        // Enable remaining temperature controls
        nott_t_ctrls.tc_sidecar.M_SetEnable();
        nott_t_ctrls.tc_photonic_chip.M_SetEnable();
        nott_t_ctrls.tc_base_plate.M_SetEnable();
        nott_t_ctrls.tc_shields.M_SetEnable();

        // Set warm-up setpoints
        nott_t_ctrls.tc_detector.M_Set_SetPoint(
            m_eSetpointType    := E_METIS_CTRL_SETPOINT_SWITCH.FIXED,
            m_lrFixedSetpoint  := cfg.lrTemp_Det,
            m_lrSetpointOffset := 0.0,
            m_pSetpointTemp    := nott_temps.M_SetTemperatureSensor(0)
        );

        nott_t_ctrls.tc_detector_spare.M_Set_SetPoint(
            m_eSetpointType    := E_METIS_CTRL_SETPOINT_SWITCH.FIXED,
            m_lrFixedSetpoint  := cfg.lrTemp_Det,
            m_lrSetpointOffset := 0.0,
            m_pSetpointTemp    := nott_temps.M_SetTemperatureSensor(0)
        );

        nott_t_ctrls.tc_sidecar.M_Set_SetPoint(
            m_eSetpointType    := E_METIS_CTRL_SETPOINT_SWITCH.FIXED,
            m_lrFixedSetpoint  := cfg.lrTemp_Sidecar,
            m_lrSetpointOffset := 0.0,
            m_pSetpointTemp    := nott_temps.M_SetTemperatureSensor(0)
        );

        nott_t_ctrls.tc_photonic_chip.M_Set_SetPoint(
            m_eSetpointType    := E_METIS_CTRL_SETPOINT_SWITCH.FIXED,
            m_lrFixedSetpoint  := cfg.lrTemp_PhotonicChip, 
            m_lrSetpointOffset := 0.0,
            m_pSetpointTemp    := nott_temps.M_SetTemperatureSensor(0)
        );

        nott_t_ctrls.tc_base_plate.M_Set_SetPoint(
            m_eSetpointType    := E_METIS_CTRL_SETPOINT_SWITCH.FIXED,
            m_lrFixedSetpoint  := cfg.lrTemp_BasePlate,
            m_lrSetpointOffset := 0.0,
            m_pSetpointTemp    := nott_temps.M_SetTemperatureSensor(0)
        );

        nott_t_ctrls.tc_shields.M_Set_SetPoint(
            m_eSetpointType    := E_METIS_CTRL_SETPOINT_SWITCH.FIXED,
            m_lrFixedSetpoint  := cfg.lrTemp_Shield,
            m_lrSetpointOffset := 0.0,
            m_pSetpointTemp    := nott_temps.M_SetTemperatureSensor(0)
        );

        stat.sState  := 'WARMING UP';
        stat.sStatus := 'Warm-up heaters enabled';

        stat.nState := E_NOTT_CRYO_WARMUP_STATE.WARMING_UP;


    E_NOTT_CRYO_WARMUP_STATE.WARMING_UP:

        out_bPermit_Evacuation_Stop := FALSE;
        out_bPermit_CoolDown        := FALSE;

        IF NOT in_bEnable THEN
            stat.nState := E_NOTT_CRYO_WARMUP_STATE.STOP_WARMUP;

        ELSIF nott_temps.out_bHighestTempValid
              AND (nott_temps.out_lrHighestTemp > cfg.lrTemp_HighLimit) THEN

            stat.bError := TRUE;
            stat.sErrorText := CONCAT('High temperature limit exceeded at ', nott_temps.out_sHighestTempName);
            stat.sStatus := stat.sErrorText;
            stat.nState := E_NOTT_CRYO_WARMUP_STATE.STOP_WARMUP;

        ELSIF bAllWarm THEN
            stat.nState := E_NOTT_CRYO_WARMUP_STATE.WARM_TEMPERATURE_ACHIEVED;
            stat.sStatus := 'Warm temperature achieved';

        ELSE
            stat.sStatus := 'Warming up...';
        END_IF;


    E_NOTT_CRYO_WARMUP_STATE.WARM_TEMPERATURE_ACHIEVED:

        IF in_bEnable THEN
            stat.sState  := 'WARM';
            stat.sStatus := 'Warm temperature achieved';

            out_bPermit_Evacuation_Stop := TRUE;
            out_bPermit_CoolDown        := TRUE;

            // Keep temperature control active at warm targets
        ELSE
            stat.nState := E_NOTT_CRYO_WARMUP_STATE.STOP_WARMUP;
        END_IF;


    E_NOTT_CRYO_WARMUP_STATE.STOP_WARMUP:

        out_bPermit_Evacuation_Stop := FALSE;
        out_bPermit_CoolDown        := FALSE;

        nott_heaters.h_detector.M_SetDisable();
        nott_heaters.h_detector_spare.M_SetDisable();
        nott_heaters.h_sidecar.M_SetDisable();
        nott_heaters.h_photonic_chip.M_SetDisable();
        nott_heaters.h_base_plate.M_SetDisable();
        nott_heaters.h_shield.M_SetDisable();

        nott_t_ctrls.tc_detector.M_SetDisable();
        nott_t_ctrls.tc_detector_spare.M_SetDisable();
        nott_t_ctrls.tc_sidecar.M_SetDisable();
        nott_t_ctrls.tc_photonic_chip.M_SetDisable();
        nott_t_ctrls.tc_base_plate.M_SetDisable();
        nott_t_ctrls.tc_shields.M_SetDisable();

        stat.bActive := FALSE;
        stat.sState  := 'OFF';
        stat.sStatus := 'Warm-up stopped';

        stat.nState := E_NOTT_CRYO_WARMUP_STATE.OFF;


ELSE
    stat.bError := TRUE;
    stat.sErrorText := 'Unknown warm-up state';
    stat.sStatus := stat.sErrorText;
    stat.nState := E_NOTT_CRYO_WARMUP_STATE.NONE;
END_CASE;

M_StateMachine := TRUE;
END_METHOD

METHOD M_UpdateStatus : BOOL
VAR_INPUT
END_VAR
stat.bEnabled		:= in_bEnable;
END_METHOD

END_FUNCTION_BLOCK

// ---- POUs/Routines/Evacuation/FB_NOTT_CRYO_EVAC.TcPOU
FUNCTION_BLOCK FB_NOTT_CRYO_EVAC EXTENDS FB_CRYO_EVAC_BASE_50
VAR_INPUT
END_VAR
VAR
	//
	// Pumps
	//
	{attribute 'TcHmiSymbol.Show'}
	pump_pvp:	FB_NOTT_PUMP_HICUBE_80_NEO;	// Pre-vacuum Pump
	{attribute 'TcHmiSymbol.Show'}
	pump_tmp:	FB_NOTT_PUMP_HIPACE80;	// Turbo Molecular Pump
	
	{attribute 'TcHmiSymbol.Show'}
	bPermitStart:	BOOL := FALSE;
	{attribute 'TcHmiSymbol.Show'}
	bPermitStop:	BOOL := FALSE;
	{attribute 'TcHmiSymbol.Show'}
	{attribute 'TcHmiSymbol.ReadOnly'}	
	bEvacuationActive:		BOOL := FALSE;			// Flag if controller is ACTIVE
	{attribute 'TcHmiSymbol.Show'}
	{attribute 'TcHmiSymbol.ReadOnly'}	
	bEmergency:		BOOL := FALSE;			// Vacuum Emergency
	
	// Power for pressure sensors (TODO)
	q_bPower_VAG1	AT %Q*:	BOOL := TRUE;
	q_bPower_VAGC	AT %Q*:	BOOL := TRUE;
	
	// Control via DIs for Pumps (DI access request)
	q_bDIsCtrl_PVP	AT %Q*:	BOOL := TRUE;
	q_bDIsCtrl_TMP	AT %Q*:	BOOL := TRUE;
	
	// Rotation speed setting mode for pumps (DI1)
	q_bRotSpeedMode_PVP	AT %Q*:	BOOL := TRUE;
	q_bRotSpeedMode_TMP	AT %Q*:	BOOL := TRUE;
	
	// Pressure valve PVV1 power
	q_bPower_PVV1	AT %Q*:	BOOL := TRUE;
	// Pressure valve PVV1 OFF Flag
	q_bPVV1_OFF_Flag	AT %Q*:	BOOL := TRUE;

	// Testing
	sDevId:	STRING := '001';
	bUpdateCmds_PVP:	BOOL;
	bUpdateCmds_TMP:	BOOL;

// NOTT-specific evacuation pressure-rise safety
tonPressureRiseWindow: TON;
bPressureRiseWindowInit: BOOL := FALSE;
bPressureRiseEvacRestarted: BOOL := FALSE;
lrPressureRiseStart: LREAL := 0.0;
lrPressureRiseDelta: LREAL := 0.0;
bPressureRiseSafetyArmed: BOOL := FALSE;
	
END_VAR

SUPER^();

// M_Configure();

// Testing: to be removed
//
// Change pump RS-485 Device ID on the fly.
M_UpdatePumpCommands();

// M_ExecuteControllers();

q_bPVV1_OFF_Flag := NOT PVV1.Actuator.q_bCtrl;

CASE stat.nState	OF
		E_CRYO_EVAC_STATE_50.NONE:
			bEvacuationActive	:= FALSE;
		
		E_CRYO_EVAC_STATE_50.OFF:
			bEvacuationActive	:= FALSE;
	ELSE
		
		bEvacuationActive		:= TRUE;
END_CASE

METHOD M_Configure
VAR_INPUT
END_VAR
VAR
	tpCfgRef:	REFERENCE TO T_NOTT_PUMP_HIPACE80_CFG;
END_VAR
//
// Specific PDS IR Imager configuration.
//
IF NOT stat.bConfigured	THEN
	//
	// MANDATORY !!!
	// Call base FB::M_Configure() to set the pointers.
	//
	SUPER^.M_Configure();
	

	// MANDATORY: Set References for pumps!!!
	// If not done, system will crash !!!
	pvpRef	REF=pump_pvp;
	tmpRef	REF=pump_tmp;
	

	// Specific instance configuration, e.g. anything different
	// from the default values given in the cfg structure 
	// of type T_CRYO_EVAC_CFG_50.
	//
	// Set pressure sensor type
	cfg.nType_VAG1	:= E_CRYO_SENSOR_TYPE_PRESS.PKR_360;
	
	// Set pressure threshold for starting TMP after opening PVV1.
	
	cfg.lrThld_TMP_after_PVV1	:= 4.8;	
	
	// Set timeout for stopping turbo pump to 15 min (900000 ms)
	tpCfgRef	REF=pump_tmp.cfg;
	tpCfgRef.nTimeoutStart	:= 900000;
	tpCfgRef.nTimeoutStop	:= 900000;


	stat.bConfigured	:= TRUE;
END_IF
END_METHOD

METHOD M_ExecuteControllers
VAR_INPUT
END_VAR
//
// Specific PDS IR Imager HW.
//

// Roughing Pump
ctrl.cor_PVP(in_bEnable:=ctrl.bEnable_PVP);	// Command override

pump_pvp(	
	in_bSimulation	:= FALSE,
	in_sName		:= 'PVP',
	in_bEnable		:= ctrl.cor_PVP.out_bEnable,
	in_nModel		:= 30,
	in_bAutoMonitor	:= TRUE,
	in_sCmdSuffix:= '$R',
	in_sReplySuffix:= '$R',
	in_nPeriod		:= 3000);

// Turbo Molecular Pump
ctrl.cor_TMP(in_bEnable:=ctrl.bEnable_TMP);	// Command override

pump_tmp(	
	in_bSimulation	:= FALSE,
	in_sName		:= 'TMP',
	in_bEnable		:= ctrl.cor_TMP.out_bEnable,
	in_nModel		:= 30,
	in_bAutoMonitor	:= TRUE,
	in_nPeriod		:= 3000,
	in_sCmdSuffix:= '$R',
	in_sReplySuffix:= '$R');


// Valves are controlled in the base FB
SUPER^.M_ExecuteControllers();
END_METHOD

METHOD M_PermitStart_Evacuation
VAR_INPUT
	in_bPermissionStart: BOOL;
END_VAR
bPermitStart := in_bPermissionStart;
END_METHOD

METHOD M_PermitStop_Evacuation
VAR_INPUT
	in_bPermissionStop: BOOL;
END_VAR
bPermitStop := in_bPermissionStop;
END_METHOD

METHOD M_SafetyCheck
VAR_INPUT
END_VAR
VAR CONSTANT
    lrPress_EmergencyReset : LREAL := 10.0E-1; // [mbar]
    lrPressRiseTrip        : LREAL := 5.0;     // [mbar rise in 10 seconds]
    tPressureRiseWindow    : TIME  := T#10S;
END_VAR
SUPER^.M_SafetyCheck();

IF NOT in_RefVAGC.stat.bValid THEN
    tonPressureRiseWindow(IN := FALSE);
    bPressureRiseWindowInit := FALSE;
    RETURN;
END_IF

// Arm this safety only after evacuation has once reached vacuum.
// This avoids false trips from noisy atmospheric-pressure readings.
IF NOT bPressureRiseSafetyArmed THEN
    tonPressureRiseWindow(IN := FALSE);
    bPressureRiseWindowInit := FALSE;

    IF bEvacuationActive
       AND (in_RefVAGC.stat.lrPressure < lrPress_EmergencyReset) THEN
        bPressureRiseSafetyArmed := TRUE;
    END_IF

    RETURN;
END_IF

// Emergency latch behavior.
IF stat.bEmergency THEN
    ctrl.bEnable_PVV1 := FALSE;
    stat.bWarning     := TRUE;

    IF in_RefVAGC.stat.lrPressure < lrPress_EmergencyReset THEN
        stat.bEmergency := FALSE;
        stat.bWarning   := FALSE;

        bPressureRiseEvacRestarted := FALSE;
        bPressureRiseWindowInit    := FALSE;
        tonPressureRiseWindow(IN := FALSE);

        // Keep armed, because we are still below the reset pressure.
        bPressureRiseSafetyArmed := TRUE;

        stat.sStatus := 'VAGC pressure below emergency reset threshold.';
    END_IF

    RETURN;
END_IF

// Normal armed monitoring.
IF NOT bPressureRiseWindowInit THEN
    lrPressureRiseStart := in_RefVAGC.stat.lrPressure;
    lrPressureRiseDelta := 0.0;
    bPressureRiseWindowInit := TRUE;
END_IF

tonPressureRiseWindow(IN := TRUE, PT := tPressureRiseWindow);

IF tonPressureRiseWindow.Q THEN
    lrPressureRiseDelta :=
        in_RefVAGC.stat.lrPressure - lrPressureRiseStart;

    IF (lrPressureRiseDelta >= lrPressRiseTrip)
       AND NOT bPressureRiseEvacRestarted THEN

        ctrl.bEnable_PVV1 := FALSE;

        stat.bEmergency := TRUE;
        stat.bWarning   := TRUE;

        bPressureRiseEvacRestarted := TRUE;

        // Replace with the correct base restart state.
        stat.nState := E_CRYO_EVAC_STATE_50.CLOSE_PVV1_START;

        stat.sStatus :=
            'Emergency: VAGC pressure rise > 5 mbar in 10 s. PVV1 closed, evacuation restarted.';
    END_IF

    IF NOT stat.bEmergency THEN
        tonPressureRiseWindow(IN := FALSE);
        bPressureRiseWindowInit := FALSE;
    END_IF
END_IF
END_METHOD

METHOD M_UpdatePumpCommands
VAR_INPUT
END_VAR
VAR
	i:			INT;
	refCfg:		REFERENCE TO T_CRYO_PUMP_SERIAL_CFG;
	refPump:	REFERENCE TO FB_CRYO_PUMP_SERIAL;
	strTmp:		STRING;	// New command string
	sCmd:		STRING;
END_VAR
IF bUpdateCmds_PVP  OR  bUpdateCmds_TMP THEN
	IF bUpdateCmds_PVP  THEN
		bUpdateCmds_PVP	:= FALSE;
		refCfg	REF=pump_pvp.cfg;
		refPump	REF=pump_pvp;
	ELSIF bUpdateCmds_TMP THEN
		bUpdateCmds_TMP	:= FALSE;
		refCfg	REF=pump_tmp.cfg;
		refPump	REF=pump_tmp;
	END_IF

	
	// Replace Device ID (first three chars) all INIT and READ commands.
	// NOTE: Commands already contain checksum in last 3 char.
	// We start from new Dev ID in the first 3 char and discard last 3 char.
	// Call to M_PVP_Checksum() will add the new checksum.
	// Skip empty commands
	FOR i:=1 TO 8 DO
		strTmp	:= sDevId;	// Start from the new ID that occupy 3 chars.
		sCmd	:= refCfg.cmdList_Init[i].cmd;
		IF sCmd <> '' THEN
			strTmp	:= CONCAT(strTmp, MID(sCmd, LEN(sCmd)-6, 4));
			refCfg.cmdList_Init[i].cmd	:= refPump.M_PVP_Checksum(strTmp);
		ELSE
			EXIT;
		END_IF
	END_FOR
	
	FOR i:=1 TO 16 DO
		strTmp	:= sDevId;	// Start from the new ID that occupy 3 chars.
		sCmd	:= refCfg.cmdList_Read[i].cmd;
		IF sCmd <> '' THEN
			strTmp	:= CONCAT(strTmp, MID(sCmd, LEN(sCmd)-6, 4));
			refCfg.cmdList_Read[i].cmd	:= refPump.M_PVP_Checksum(strTmp);
		ELSE
			EXIT;
		END_IF
	END_FOR
	
END_IF
END_METHOD

END_FUNCTION_BLOCK

// ---- POUs/Devices/ThermalBox/FB_NOTT_THERMAL_BOX_CONTROL.TcPOU
FUNCTION_BLOCK FB_NOTT_THERMAL_BOX_CONTROL
VAR_INPUT
	in_tCycleTime:	TIME := T#10MS;
END_VAR
VAR_IN_OUT
	{attribute 'OPC.UA.DA' := '0'}
	nott_temps:						FB_NOTT_TEMPERATURES;
	{attribute 'OPC.UA.DA' := '0'}
	nott_heaters:					FB_NOTT_HEATERS;
	{attribute 'OPC.UA.DA' := '0'}
	nott_t_ctrls:      				FB_NOTT_TCTRLs;
	{attribute 'OPC.UA.DA' := '0'}
	nott_t_votes: 					FB_NOTT_VOTERS;
END_VAR
VAR
// 	{attribute 'TcHmiSymbol.Show'}
// 	cfg:	T_NOTT_THERMAL_BOX_CFG;
// 	{attribute 'TcHmiSymbol.Show'}
// 	ctrl:	T_NOTT_THERMAL_BOX_CTRL;
// 	{attribute 'TcHmiSymbol.Show'}
// 	stat:	T_NOTT_THERMAL_BOX_STAT;

	{attribute 'TcHmiSymbol.Show'}
	tc_fan:		FB_NOTT_CTRL_TEMPERATURE;
	{attribute 'TcHmiSymbol.Show'}
	tc_valve:	FB_NOTT_CTRL_TEMPERATURE;
	{attribute 'TcHmiSymbol.Show'}
	fan:		FB_NOTT_FAN;
	{attribute 'TcHmiSymbol.Show'}
	valve:		FB_METIS_CONTROL_VALVE;

	bFanAutoReady:		BOOL;
	bValveAutoReady:	BOOL;
END_VAR

METHOD M_SetDisable
//ctrl.bEnable := FALSE;
END_METHOD

METHOD M_SetEnable
//ctrl.bEnable := TRUE;
END_METHOD

END_FUNCTION_BLOCK

// ---- POUs/Devices/Fans/FB_NOTT_FAN.TcPOU
FUNCTION_BLOCK FB_NOTT_FAN
VAR_INPUT
	in_sName:				STRING;
	in_sAutoSetpointSource:	STRING;
	in_lrAutoSetpointValue:	LREAL;		// Temperature-controller output [0..100 %]
	in_tCycleTime:			TIME := T#10MS;
END_VAR
VAR
	{attribute 'TcHmiSymbol.Show'}
	cfg:	T_NOTT_FAN_CFG;
	{attribute 'TcHmiSymbol.Show'}
	ctrl:	T_NOTT_FAN_CTRL;
	{attribute 'TcHmiSymbol.Show'}
	stat:	T_NOTT_FAN_STAT;

	// Link these process-image variables to the selected EL2535 and ES1084 channels.
	{attribute 'TcHmiSymbol.Show'}
	i_bTach AT %I*:	BOOL;
	{attribute 'TcHmiSymbol.Show'}
	q_nPwmCommand AT %Q*:	INT;

	rtrigTach:	R_TRIG;
	rtrigEnable:	R_TRIG;
	tonRpmWindow:	TON;
	tonNoTach:	TON;
	tonStartBoost:	TON;
	bStarting:	BOOL := FALSE;
	bTach:		BOOL := FALSE;
	lrDemand:	LREAL := 0.0;
	lrOutputDuty:	LREAL := 0.0;
	nWindowPulses:	UDINT := 0;
END_VAR

stat.sName := in_sName;
stat.sAutoSetpointSource := in_sAutoSetpointSource;

// The thermal-box controller must be configured reverse acting (negative Kp):
// fan demand increases when measured temperature rises above setpoint.
IF ctrl.bAuto THEN
	lrDemand := in_lrAutoSetpointValue;
ELSE
	lrDemand := ctrl.lrManualDutyPct;
END_IF

IF lrDemand < 0.0 THEN
	lrDemand := 0.0;
ELSIF lrDemand > 100.0 THEN
	lrDemand := 100.0;
END_IF
stat.lrDemandPct := lrDemand;

rtrigEnable(CLK := ctrl.bEnable AND (lrDemand > 0.0));
IF rtrigEnable.Q THEN
	bStarting := TRUE;
	tonStartBoost(IN := FALSE, PT := cfg.tStartBoost);
END_IF

IF NOT ctrl.bEnable OR (lrDemand <= 0.0) THEN
	bStarting := FALSE;
	tonStartBoost(IN := FALSE, PT := cfg.tStartBoost);
	stat.lrDutyPct := 0.0;
	stat.bActive := ctrl.bEnable;
ELSE
	stat.bActive := TRUE;

	IF bStarting THEN
		tonStartBoost(IN := TRUE, PT := cfg.tStartBoost);
		stat.lrDutyPct := cfg.lrStartDutyPct;
		IF tonStartBoost.Q THEN
			bStarting := FALSE;
			tonStartBoost(IN := FALSE, PT := cfg.tStartBoost);
		END_IF
	ELSE
		IF lrDemand <= 0.0 THEN
			stat.lrDutyPct := 0.0;
		ELSIF lrDemand < cfg.lrMinRunningDutyPct THEN
			stat.lrDutyPct := cfg.lrMinRunningDutyPct;
		ELSIF lrDemand > cfg.lrMaxDutyPct THEN
			stat.lrDutyPct := cfg.lrMaxDutyPct;
		ELSE
			stat.lrDutyPct := lrDemand;
		END_IF
	END_IF
END_IF

IF stat.lrDutyPct < 0.0 THEN
	stat.lrDutyPct := 0.0;
ELSIF stat.lrDutyPct > 100.0 THEN
	stat.lrDutyPct := 100.0;
END_IF

lrOutputDuty := stat.lrDutyPct;
IF cfg.bInvertPwmOutput THEN
	lrOutputDuty := 100.0 - lrOutputDuty;
END_IF
q_nPwmCommand := LREAL_TO_INT(lrOutputDuty * INT_TO_LREAL(cfg.nPwmFullScale) / 100.0);

// ES1084 tach input. The fan supplies two rising pulses per revolution.
bTach := i_bTach;
IF cfg.bInvertTachInput THEN
	bTach := NOT bTach;
END_IF
rtrigTach(CLK := bTach);

IF rtrigTach.Q THEN
	nWindowPulses := nWindowPulses + 1;
	stat.nPulseCount := stat.nPulseCount + 1;
END_IF

tonRpmWindow(IN := TRUE, PT := cfg.tRpmWindow);
IF tonRpmWindow.Q THEN
	IF cfg.nPulsesPerRevolution > 0 THEN
		stat.lrSpeedRpm :=
			UDINT_TO_LREAL(nWindowPulses) * 60.0
			/ UINT_TO_LREAL(cfg.nPulsesPerRevolution)
			/ (TIME_TO_LREAL(cfg.tRpmWindow) / 1000.0);
	ELSE
		stat.lrSpeedRpm := 0.0;
	END_IF
	nWindowPulses := 0;
	tonRpmWindow(IN := FALSE, PT := cfg.tRpmWindow);
END_IF

// Reset the no-tach timer on every observed pulse.
tonNoTach(
	IN := ctrl.bEnable
		AND (stat.lrDutyPct >= cfg.lrMinRunningDutyPct)
		AND NOT rtrigTach.Q,
	PT := cfg.tStallDelay);

stat.bStallAlarm := tonNoTach.Q;
stat.bRunning := ctrl.bEnable AND (stat.lrSpeedRpm > 0.0) AND NOT stat.bStallAlarm;

// At maximum fan speed the pulse period is about 7 ms. A 10 ms task can miss
// edges even before considering the ES1084 3 ms input filter.
stat.bTachMeasurementLimited := in_tCycleTime > T#2MS;

METHOD M_SetDisable
ctrl.bEnable := FALSE;
END_METHOD

METHOD M_SetEnable
ctrl.bEnable := TRUE;
END_METHOD

END_FUNCTION_BLOCK

// ---- GlobalTextList.TcGTLO
TEXTLIST GlobalTextList
  876 = '%.1f'
  866 = '%.2f'
  778 = '%d'
  154 = '%s'
  640 = 'Configuration'
  284 = 'Control Mode'
  439 = 'Ctrl Signal :'
  784 = 'Drive Elec. Hours :'
  133 = 'Drive Elec. Temp [°C] :'
  905 = 'Error :'
  325 = 'Error Status'
  386 = 'Failure/Error Core'
  837 = 'FW Version'
  1833 = 'FW Version :'
  981 = 'Gas Balast Valve'
  418 = 'Gas Ballast Valve Enable'
  116 = 'Gas Ballast valve status'
  110 = 'GroupBox'
  858 = 'HW Version'
  2127 = 'HW Version :'
  873 = 'ID'
  145 = 'If ON, control output signal is active.'
  81 = 'Initialized'
  257 = 'Motor Current [mA] :'
  157 = 'Motor Power [W] :'
  804 = 'Motor Voltage [V] :'
  396 = 'Nominal Speed [rpm] :'
  611 = 'OK for Process, i.e. speed ≥ nominal speed'
  413 = 'presence of a warning'
  172 = 'Pressure'
  186 = 'Pressure Gauge'
  407 = 'Pressure Raw '
  894 = 'Pressure Sensor '
  216 = 'Pressure Sensor Active'
  434 = 'Pressure Sensor ON'
  587 = 'Pressure Text'
  385 = 'Pump Hours :'
  1038 = 'pump speed > 0 rpm'
  1651 = 'Pump Speed [rpm] :'
  148 = 'Pump State'
  1668 = 'Pump Temp [°C] :'
  384 = 'Ready :'
  12 = 'Running :'
  16 = 'Sensor Failed'
  670 = 'Sensor State'
  19 = 'START'
  401 = 'Status'
  119 = 'STOP'
  935 = 'Venting Enable'
END_TEXTLIST

// ---- VISUs/GUI_TEMPLATE_HIPACE_80.TcVIS
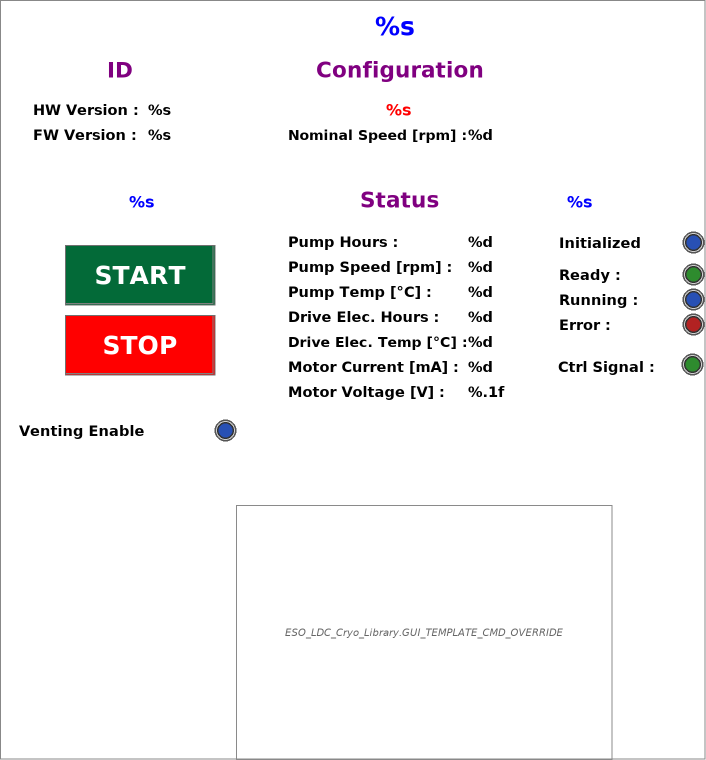
VISUALIZATION GUI_TEMPLATE_HIPACE_80  // 706x760
VAR_IN_OUT
	m_Instance:	FB_NOTT_PUMP_HIPACE80;
	m_bEnable:	BOOL;	// Flag to start/stop the pump
END_VAR
    Rectangle (45,55 150x30), "ID"
    Rectangle (310,55 180x30), "Configuration"
    Rectangle (325,185 150x30), "Status"
    Lamp1 (681,262 25x25), tooltip "OK for Process, i.e. speed ≥ nominal speed", variable: m_Instance.stat.bReady, style: Lamp-Lamp1-Green
    Lamp1 (681,287 25x25), tooltip "pump speed > 0 rpm", variable: m_Instance.stat.bMoving, style: Lamp-Lamp1-Blue
    Lamp1 (681,312 25x25), tooltip "presence of a warning", variable: m_Instance.stat.bFailure, style: Lamp-Lamp1-Red
    Rectangle (556,260 110x30), "Ready :"
    Rectangle (556,285 110x30), "Running :"
    Rectangle (556,310 110x30), "Error :"
    Rectangle (285,120 180x30), "Nominal Speed [rpm] :"
    Rectangle (285,227 180x30), "Pump Hours :"
    Rectangle (285,302 180x30), "Drive Elec. Hours :"
    Rectangle (465,120 70x30), "%d", text variable: m_Instance.stat.nNominalSpeed
    Rectangle (465,227 70x30), "%d", text variable: m_Instance.stat.nPumpHours
    Rectangle (465,302 70x30), "%d", text variable: m_Instance.stat.nElecHours
    Rectangle (285,252 180x30), "Pump Speed [rpm] :"
    Rectangle (465,252 70x30), "%d", text variable: m_Instance.stat.nPumpSpeed
    Rectangle (285,327 180x30), "Drive Elec. Temp [°C] :", text variable: m_Instance.stat.nElecTemp
    Rectangle (465,327 70x30), "%d", text variable: m_Instance.stat.nElecTemp
    Rectangle (285,277 180x30), "Pump Temp [°C] :"
    Rectangle (465,277 70x30), "%d", text variable: m_Instance.stat.nPumpTemp
    Rectangle (285,352 180x30), "Motor Current [mA] :", text variable: m_Instance.stat.nMotorCurr
    Rectangle (465,352 70x30), "%d", text variable: m_Instance.stat.nMotorCurr
    Rectangle (285,377 180x30), "Motor Voltage [V] :", text variable: m_Instance.stat.nMotorVolt
    Rectangle (465,377 70x30), "%.1f", text variable: m_Instance.stat.lrMotorVolt
    Rectangle (280,11 230x30), "%s", text variable: m_Instance.in_sName
    Rectangle (289,95 220x30), "%s", tooltip "Control Mode", text variable: m_Instance.stat.sCtrlMode
    Rectangle (145,95 130x30), "%s", tooltip "HW Version", text variable: m_Instance.stat.sHwVersion
    Rectangle (145,120 130x30), "%s", tooltip "FW Version", text variable: m_Instance.stat.sFwVersion
    Button (65,245 150x60), "START"
        OnMouseClick: execute { m_bEnable := TRUE; }
    Button (65,315 150x60), "STOP"
        OnMouseClick: execute { m_bEnable := FALSE; }
    Lamp1 (680,352 25x25), tooltip "If ON, control output signal is active.", variable: m_Instance.q_bStart, style: Lamp-Lamp1-Green
    Rectangle (555,352 110x30), "Ctrl Signal :"
    Rectangle (457,187 246x30), "%s", tooltip "Pump State", text variable: m_Instance.stat.sPumpState
    Rectangle (92,187 100x30), "%s", tooltip "Error Status", text variable: m_Instance.stat.sFailureCode
    Rectangle (30,95 110x30), "HW Version :"
    Rectangle (30,120 110x30), "FW Version :"
    Rectangle (556,228 110x30), "Initialized"
    Lamp1 (681,230 25x25), tooltip "OK for Process, i.e. speed ≥ nominal speed", variable: m_Instance.stat.bInitialised, style: Lamp-Lamp1-Blue
    Lamp1 (213,418 25x25), tooltip "OK for Process, i.e. speed ≥ nominal speed", variable: m_Instance.stat.bVentEnable, style: Lamp-Lamp1-Blue
    Rectangle (16,416 182x30), "Venting Enable"
    Frame (236,505 376x255)
        shows ESO_LDC_Cryo_Library.GUI_TEMPLATE_CMD_OVERRIDE(m_Cmd := MAIN.nott_cryo_ctrl.evac.ctrl.cor_TMP)
END_VISUALIZATION

// ---- VISUs/TEMPLATE_NOTT_PUMPS.TcVIS
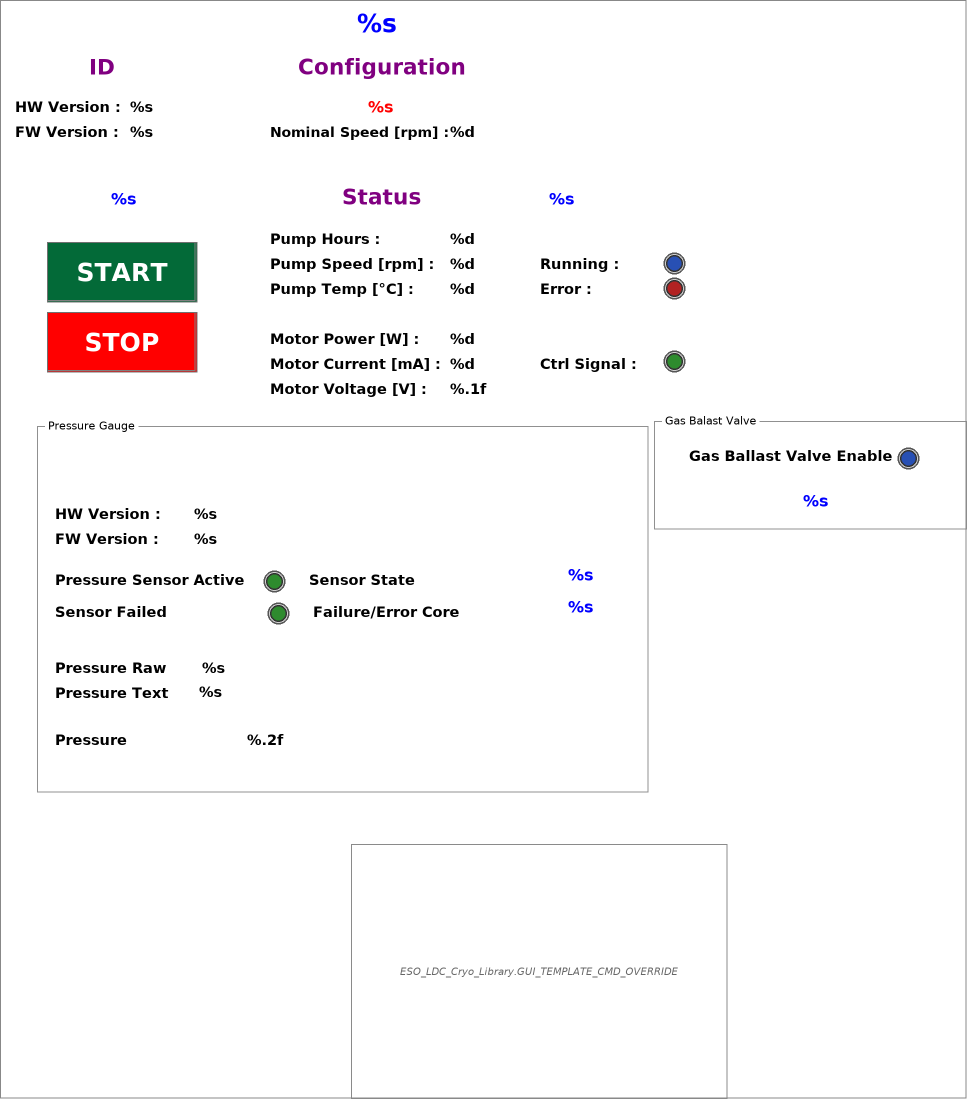
VISUALIZATION TEMPLATE_NOTT_PUMPS  // 967x1099
VAR_IN_OUT
	m_Instance:	FB_NOTT_PUMP_HICUBE_80_NEO;
	m_bEnable:	BOOL;	// Flag to start/stop the pump
	
END_VAR
    Rectangle (27,52 150x30), "ID"
    Rectangle (292,52 180x30), "Configuration"
    Rectangle (307,182 150x30), "Status"
    Lamp1 (662,251 25x25), tooltip "pump speed > 0 rpm", variable: m_Instance.stat.bMoving, style: Lamp-Lamp1-Blue
    Lamp1 (662,276 25x25), tooltip "presence of a warning", variable: m_Instance.stat.bFailure, style: Lamp-Lamp1-Red
    Rectangle (537,249 110x30), "Running :"
    Rectangle (537,274 110x30), "Error :"
    Rectangle (267,117 180x30), "Nominal Speed [rpm] :"
    Rectangle (267,224 180x30), "Pump Hours :"
    Rectangle (447,117 70x30), "%d", text variable: m_Instance.stat.nNominalSpeed
    Rectangle (447,224 70x30), "%d", text variable: m_Instance.stat.nPumpHours
    Rectangle (267,249 180x30), "Pump Speed [rpm] :"
    Rectangle (447,249 70x30), "%d", text variable: m_Instance.stat.nPumpSpeed
    Rectangle (267,274 180x30), "Pump Temp [°C] :"
    Rectangle (447,274 70x30), "%d", text variable: m_Instance.stat.nPumpTemp
    Rectangle (267,349 180x30), "Motor Current [mA] :"
    Rectangle (447,349 70x30), "%d", text variable: m_Instance.stat.nMotorCurr
    Rectangle (267,374 180x30), "Motor Voltage [V] :"
    Rectangle (447,374 70x30), "%.1f", text variable: m_Instance.stat.lrMotorVolt
    Rectangle (262,8 230x30), "%s", text variable: m_Instance.in_sName
    Rectangle (271,92 220x30), "%s", tooltip "Control Mode", text variable: m_Instance.stat.sCtrlViaInt
    Rectangle (127,92 130x30), "%s", tooltip "HW Version", text variable: m_Instance.stat.sHwVersion
    Rectangle (127,117 130x30), "%s", tooltip "FW Version", text variable: m_Instance.stat.sFwVersion
    Button (47,242 150x60), "START"
        OnMouseClick: execute { m_bEnable := TRUE; }
    Button (47,312 150x60), "STOP"
        OnMouseClick: execute { m_bEnable := FALSE; }
    Lamp1 (662,349 25x25), tooltip "If ON, control output signal is active.", variable: m_Instance.q_bStart, style: Lamp-Lamp1-Green
    Rectangle (537,349 110x30), "Ctrl Signal :"
    Rectangle (439,184 246x30), "%s", tooltip "Pump State", text variable: m_Instance.stat.sPumpState
    Rectangle (74,184 100x30), "%s", tooltip "Error Status", text variable: m_Instance.stat.sFailureCode
    Rectangle (267,324 180x30), "Motor Power [W] :"
    Rectangle (447,324 70x30), "%d", text variable: m_Instance.stat.nElecPower
    Rectangle (12,92 110x30), "HW Version :"
    Rectangle (12,117 110x30), "FW Version :"
    Frame (351,844 376x255)
        shows ESO_LDC_Cryo_Library.GUI_TEMPLATE_CMD_OVERRIDE(m_Cmd := MAIN.nott_cryo_ctrl.evac.ctrl.cor_PVP)
    GroupBox (37,418 611x374), "Pressure Gauge"
        Lamp1 (225,151 25x25), tooltip "Pressure Sensor ON", variable: m_Instance.stat.PresSens_bSensorOn, style: Lamp-Lamp1-Green
        Rectangle (15,147 254x30), "Pressure Sensor Active"
        Lamp1 (229,183 25x25), tooltip "Pressure Sensor ON", variable: m_Instance.stat.PresSens_bFailure, style: Lamp-Lamp1-Green
        Rectangle (269,147 254x30), "Sensor State"
        Rectangle (450,174 188x30), "%s", tooltip "Error Status", text variable: m_Instance.stat.PresSens_sFailureCode
        Rectangle (273,179 254x30), "Failure/Error Core"
        Rectangle (15,179 254x30), "Sensor Failed"
        Rectangle (450,142 188x30), "%s", tooltip "Error Status", text variable: m_Instance.stat.PresSens_sSensorState
        Rectangle (15,81 110x30), "HW Version :"
        Rectangle (154,81 130x30), "%s", tooltip "HW Version", text variable: m_Instance.stat.PresSens_sHwVersion
        Rectangle (154,106 130x30), "%s", tooltip "FW Version", text variable: m_Instance.stat.PresSens_sFwVersion
        Rectangle (15,106 110x30), "FW Version :"
        Rectangle (15,235 138x30), "Pressure Raw"
        Rectangle (162,235 130x30), "%s", tooltip "HW Version", text variable: m_Instance.stat.PresSens_sPressureRaw
        Rectangle (159,259 130x30), "%s", tooltip "FW Version", text variable: m_Instance.stat.PresSens_sPressureText
        Rectangle (15,260 142x30), "Pressure Text"
        Rectangle (15,307 180x30), "Pressure"
        Rectangle (207,307 197x30), "%.2f", text variable: m_Instance.stat.PresSens_lrPressure_hPa
    GroupBox (654,413 313x116), "Gas Balast Valve"
        Rectangle (39,73 246x30), "%s", tooltip "Gas Ballast valve status", text variable: m_Instance.stat.sGasBallastMode
        Lamp1 (242,33 25x25), tooltip "If ON, control output signal is active.", variable: m_Instance.stat.bGasBallastEnabled, style: Lamp-Lamp1-Blue
        Rectangle (32,28 211x30), "Gas Ballast Valve Enable"
END_VISUALIZATION

// ---- VISUs/VISU_BASE_PLATE_HTR.TcVIS
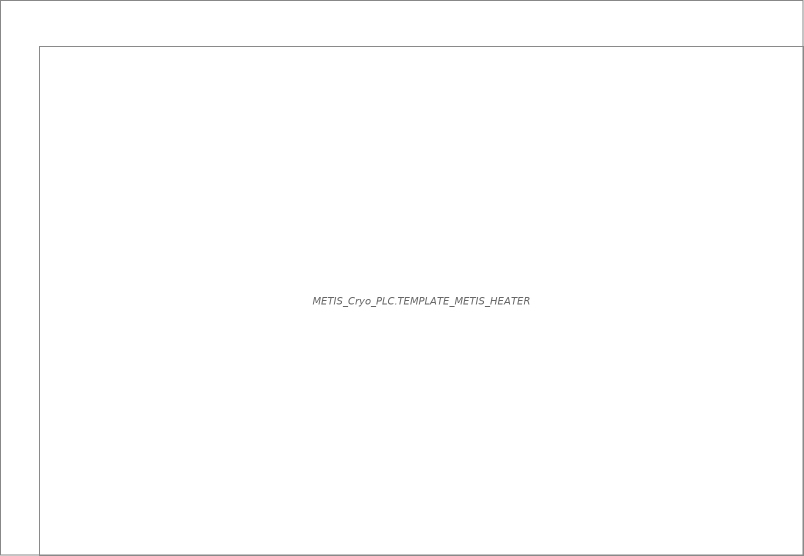
VISUALIZATION VISU_BASE_PLATE_HTR  // 804x556
    Frame (39,46 765x510)
        shows METIS_Cryo_PLC.TEMPLATE_METIS_HEATER(m_instance := MAIN.nott_cryo_ctrl.nott_heaters.h_base_plate)
END_VISUALIZATION

// ---- VISUs/VISU_Detector_Heater.TcVIS
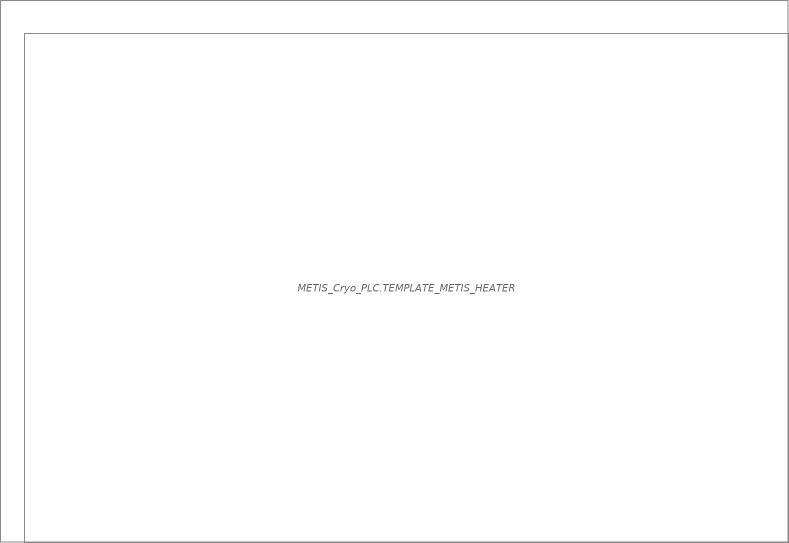
VISUALIZATION VISU_Detector_Heater  // 789x543
    Frame (24,33 765x510)
        shows METIS_Cryo_PLC.TEMPLATE_METIS_HEATER(m_instance := MAIN.nott_cryo_ctrl.nott_heaters.h_detector)
END_VISUALIZATION

// ---- VISUs/VISU_NOTT_PRESSURES.TcVIS
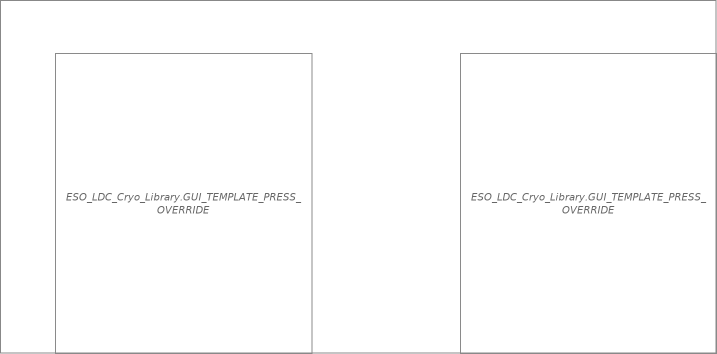
VISUALIZATION VISU_NOTT_PRESSURES  // 717x354
    Frame (55,53 257x301)
        shows ESO_LDC_Cryo_Library.GUI_TEMPLATE_PRESS_OVERRIDE(m_Cmd := MAIN.nott_cryo_ctrl.ctrl.por_VAGC, m_Press := MAIN.nott_cryo_ctrl.VAGC)
    Frame (460,53 257x301)
        shows ESO_LDC_Cryo_Library.GUI_TEMPLATE_PRESS_OVERRIDE(m_Cmd := MAIN.nott_cryo_ctrl.ctrl.por_HPG, m_Press := MAIN.nott_cryo_ctrl.HPG)
END_VISUALIZATION

// ---- VISUs/VISU_NOTT_RP.TcVIS
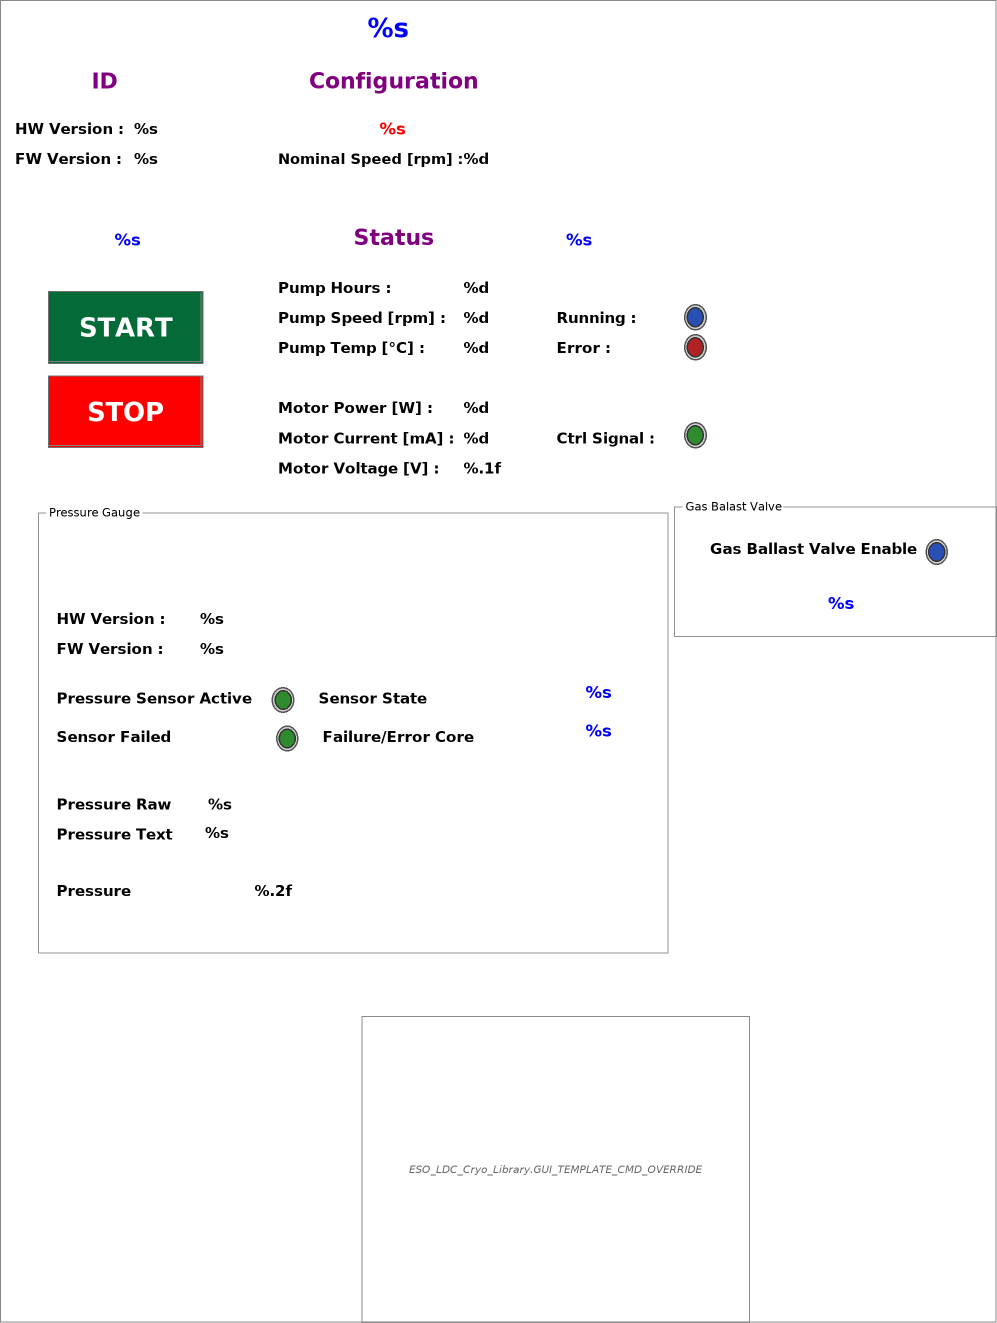
VISUALIZATION VISU_NOTT_RP  // 997x1323
    Frame (0,0 997x1323)
        shows TEMPLATE_NOTT_PUMPS(m_Instance := MAIN.nott_cryo_ctrl.evac.pump_pvp)
END_VISUALIZATION

// ---- VISUs/VISU_NOTT_TP.TcVIS
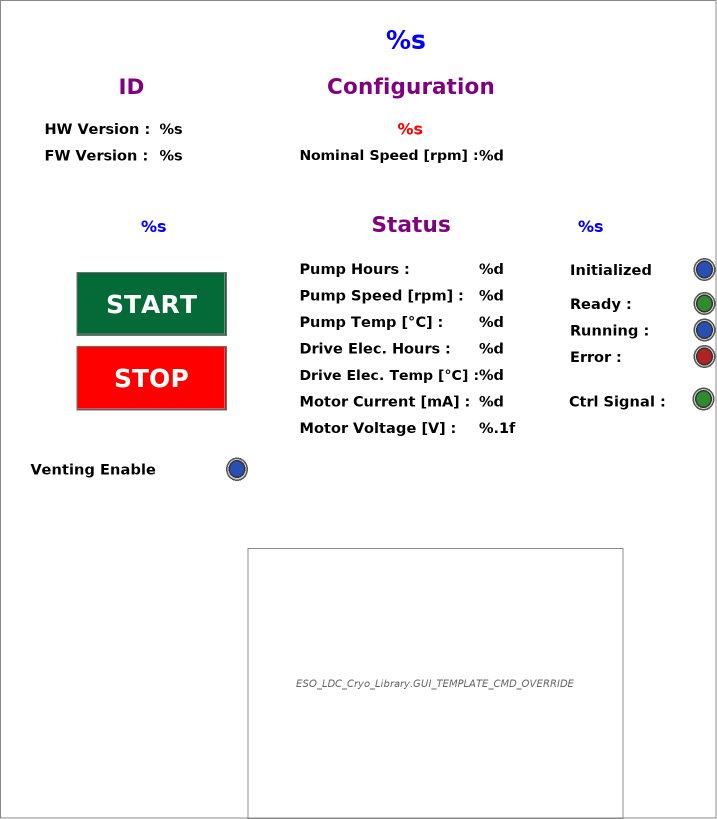
VISUALIZATION VISU_NOTT_TP  // 717x819
    Frame (12,12 705x807)
        shows GUI_TEMPLATE_HIPACE_80(m_Instance := MAIN.nott_cryo_ctrl.evac.pump_tmp)
END_VISUALIZATION

// ---- VISUs/VISU_PTC_COOLER.TcVIS
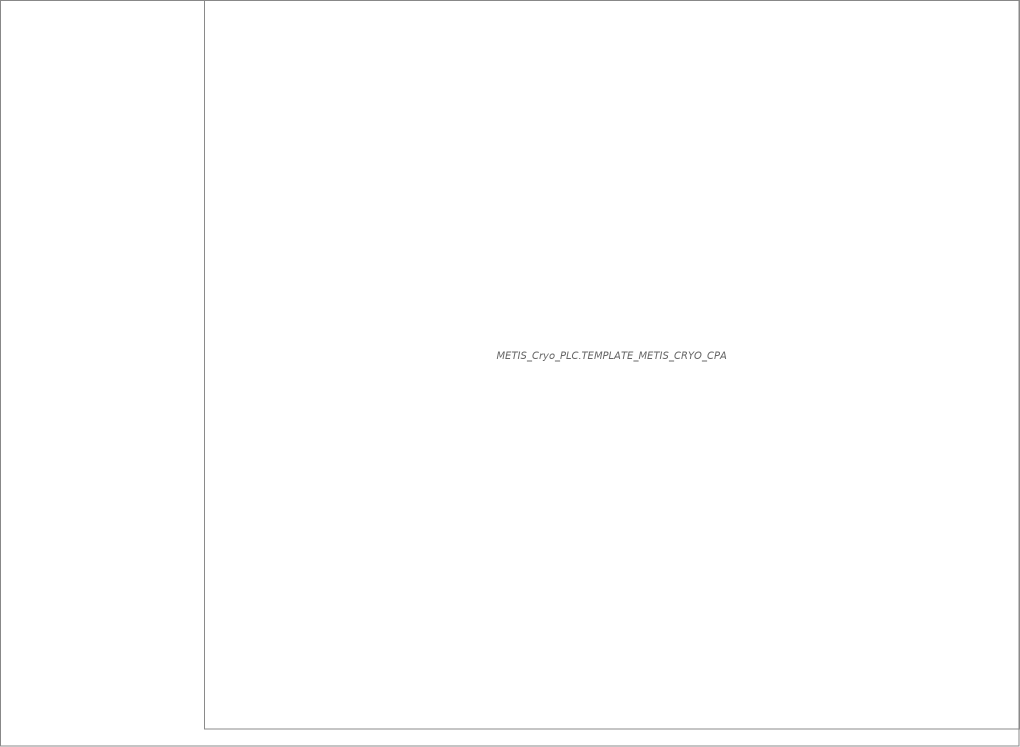
VISUALIZATION VISU_PTC_COOLER  // 1020x747
    Frame (204,-18 816x747)
        shows METIS_Cryo_PLC.TEMPLATE_METIS_CRYO_CPA(m_Instance := MAIN.nott_cryo_ctrl.cooler, m_Cmd := MAIN.nott_cryo_ctrl.ctrl.cor_Cooler)
END_VISUALIZATION
